    PROC LoadSlot_P06(num slot, VAR bool used, VAR num subType, VAR num toolSel, VAR num lenMM,
                       VAR robtarget arcStart, VAR robtarget arcEnd, VAR robtarget approach, VAR robtarget retract, VAR robtarget trans)
        IF slot = 1 THEN
            used := P06W01_Used;
            subType := P06W01_SubType;
            toolSel := P06W01_ToolSel;
            lenMM := P06W01_LenMM;
            arcStart := P06W01_ArcStart;
            arcEnd := P06W01_ArcEnd;
            approach := P06W01_Approach;
            retract := P06W01_Retract;
            trans := P06W01_Trans;
        ELSEIF slot = 2 THEN
            used := P06W02_Used;
            subType := P06W02_SubType;
            toolSel := P06W02_ToolSel;
            lenMM := P06W02_LenMM;
            arcStart := P06W02_ArcStart;
            arcEnd := P06W02_ArcEnd;
            approach := P06W02_Approach;
            retract := P06W02_Retract;
            trans := P06W02_Trans;
        ELSEIF slot = 3 THEN
            used := P06W03_Used;
            subType := P06W03_SubType;
            toolSel := P06W03_ToolSel;
            lenMM := P06W03_LenMM;
            arcStart := P06W03_ArcStart;
            arcEnd := P06W03_ArcEnd;
            approach := P06W03_Approach;
            retract := P06W03_Retract;
            trans := P06W03_Trans;
        ELSEIF slot = 4 THEN
            used := P06W04_Used;
            subType := P06W04_SubType;
            toolSel := P06W04_ToolSel;
            lenMM := P06W04_LenMM;
            arcStart := P06W04_ArcStart;
            arcEnd := P06W04_ArcEnd;
            approach := P06W04_Approach;
            retract := P06W04_Retract;
            trans := P06W04_Trans;
        ELSEIF slot = 5 THEN
            used := P06W05_Used;
            subType := P06W05_SubType;
            toolSel := P06W05_ToolSel;
            lenMM := P06W05_LenMM;
            arcStart := P06W05_ArcStart;
            arcEnd := P06W05_ArcEnd;
            approach := P06W05_Approach;
            retract := P06W05_Retract;
            trans := P06W05_Trans;
        ELSEIF slot = 6 THEN
            used := P06W06_Used;
            subType := P06W06_SubType;
            toolSel := P06W06_ToolSel;
            lenMM := P06W06_LenMM;
            arcStart := P06W06_ArcStart;
            arcEnd := P06W06_ArcEnd;
            approach := P06W06_Approach;
            retract := P06W06_Retract;
            trans := P06W06_Trans;
        ELSEIF slot = 7 THEN
            used := P06W07_Used;
            subType := P06W07_SubType;
            toolSel := P06W07_ToolSel;
            lenMM := P06W07_LenMM;
            arcStart := P06W07_ArcStart;
            arcEnd := P06W07_ArcEnd;
            approach := P06W07_Approach;
            retract := P06W07_Retract;
            trans := P06W07_Trans;
        ELSEIF slot = 8 THEN
            used := P06W08_Used;
            subType := P06W08_SubType;
            toolSel := P06W08_ToolSel;
            lenMM := P06W08_LenMM;
            arcStart := P06W08_ArcStart;
            arcEnd := P06W08_ArcEnd;
            approach := P06W08_Approach;
            retract := P06W08_Retract;
            trans := P06W08_Trans;
        ELSEIF slot = 9 THEN
            used := P06W09_Used;
            subType := P06W09_SubType;
            toolSel := P06W09_ToolSel;
            lenMM := P06W09_LenMM;
            arcStart := P06W09_ArcStart;
            arcEnd := P06W09_ArcEnd;
            approach := P06W09_Approach;
            retract := P06W09_Retract;
            trans := P06W09_Trans;
        ELSEIF slot = 10 THEN
            used := P06W10_Used;
            subType := P06W10_SubType;
            toolSel := P06W10_ToolSel;
            lenMM := P06W10_LenMM;
            arcStart := P06W10_ArcStart;
            arcEnd := P06W10_ArcEnd;
            approach := P06W10_Approach;
            retract := P06W10_Retract;
            trans := P06W10_Trans;
        ELSEIF slot = 11 THEN
            used := P06W11_Used;
            subType := P06W11_SubType;
            toolSel := P06W11_ToolSel;
            lenMM := P06W11_LenMM;
            arcStart := P06W11_ArcStart;
            arcEnd := P06W11_ArcEnd;
            approach := P06W11_Approach;
            retract := P06W11_Retract;
            trans := P06W11_Trans;
        ELSEIF slot = 12 THEN
            used := P06W12_Used;
            subType := P06W12_SubType;
            toolSel := P06W12_ToolSel;
            lenMM := P06W12_LenMM;
            arcStart := P06W12_ArcStart;
            arcEnd := P06W12_ArcEnd;
            approach := P06W12_Approach;
            retract := P06W12_Retract;
            trans := P06W12_Trans;
        ELSEIF slot = 13 THEN
            used := P06W13_Used;
            subType := P06W13_SubType;
            toolSel := P06W13_ToolSel;
            lenMM := P06W13_LenMM;
            arcStart := P06W13_ArcStart;
            arcEnd := P06W13_ArcEnd;
            approach := P06W13_Approach;
            retract := P06W13_Retract;
            trans := P06W13_Trans;
        ELSEIF slot = 14 THEN
            used := P06W14_Used;
            subType := P06W14_SubType;
            toolSel := P06W14_ToolSel;
            lenMM := P06W14_LenMM;
            arcStart := P06W14_ArcStart;
            arcEnd := P06W14_ArcEnd;
            approach := P06W14_Approach;
            retract := P06W14_Retract;
            trans := P06W14_Trans;
        ELSEIF slot = 15 THEN
            used := P06W15_Used;
            subType := P06W15_SubType;
            toolSel := P06W15_ToolSel;
            lenMM := P06W15_LenMM;
            arcStart := P06W15_ArcStart;
            arcEnd := P06W15_ArcEnd;
            approach := P06W15_Approach;
            retract := P06W15_Retract;
            trans := P06W15_Trans;
        ELSEIF slot = 16 THEN
            used := P06W16_Used;
            subType := P06W16_SubType;
            toolSel := P06W16_ToolSel;
            lenMM := P06W16_LenMM;
            arcStart := P06W16_ArcStart;
            arcEnd := P06W16_ArcEnd;
            approach := P06W16_Approach;
            retract := P06W16_Retract;
            trans := P06W16_Trans;
        ELSEIF slot = 17 THEN
            used := P06W17_Used;
            subType := P06W17_SubType;
            toolSel := P06W17_ToolSel;
            lenMM := P06W17_LenMM;
            arcStart := P06W17_ArcStart;
            arcEnd := P06W17_ArcEnd;
            approach := P06W17_Approach;
            retract := P06W17_Retract;
            trans := P06W17_Trans;
        ELSEIF slot = 18 THEN
            used := P06W18_Used;
            subType := P06W18_SubType;
            toolSel := P06W18_ToolSel;
            lenMM := P06W18_LenMM;
            arcStart := P06W18_ArcStart;
            arcEnd := P06W18_ArcEnd;
            approach := P06W18_Approach;
            retract := P06W18_Retract;
            trans := P06W18_Trans;
        ELSEIF slot = 19 THEN
            used := P06W19_Used;
            subType := P06W19_SubType;
            toolSel := P06W19_ToolSel;
            lenMM := P06W19_LenMM;
            arcStart := P06W19_ArcStart;
            arcEnd := P06W19_ArcEnd;
            approach := P06W19_Approach;
            retract := P06W19_Retract;
            trans := P06W19_Trans;
        ELSEIF slot = 20 THEN
            used := P06W20_Used;
            subType := P06W20_SubType;
            toolSel := P06W20_ToolSel;
            lenMM := P06W20_LenMM;
            arcStart := P06W20_ArcStart;
            arcEnd := P06W20_ArcEnd;
            approach := P06W20_Approach;
            retract := P06W20_Retract;
            trans := P06W20_Trans;
        ELSEIF slot = 21 THEN
            used := P06W21_Used;
            subType := P06W21_SubType;
            toolSel := P06W21_ToolSel;
            lenMM := P06W21_LenMM;
            arcStart := P06W21_ArcStart;
            arcEnd := P06W21_ArcEnd;
            approach := P06W21_Approach;
            retract := P06W21_Retract;
            trans := P06W21_Trans;
        ELSEIF slot = 22 THEN
            used := P06W22_Used;
            subType := P06W22_SubType;
            toolSel := P06W22_ToolSel;
            lenMM := P06W22_LenMM;
            arcStart := P06W22_ArcStart;
            arcEnd := P06W22_ArcEnd;
            approach := P06W22_Approach;
            retract := P06W22_Retract;
            trans := P06W22_Trans;
        ELSEIF slot = 23 THEN
            used := P06W23_Used;
            subType := P06W23_SubType;
            toolSel := P06W23_ToolSel;
            lenMM := P06W23_LenMM;
            arcStart := P06W23_ArcStart;
            arcEnd := P06W23_ArcEnd;
            approach := P06W23_Approach;
            retract := P06W23_Retract;
            trans := P06W23_Trans;
        ELSEIF slot = 24 THEN
            used := P06W24_Used;
            subType := P06W24_SubType;
            toolSel := P06W24_ToolSel;
            lenMM := P06W24_LenMM;
            arcStart := P06W24_ArcStart;
            arcEnd := P06W24_ArcEnd;
            approach := P06W24_Approach;
            retract := P06W24_Retract;
            trans := P06W24_Trans;
        ELSEIF slot = 25 THEN
            used := P06W25_Used;
            subType := P06W25_SubType;
            toolSel := P06W25_ToolSel;
            lenMM := P06W25_LenMM;
            arcStart := P06W25_ArcStart;
            arcEnd := P06W25_ArcEnd;
            approach := P06W25_Approach;
            retract := P06W25_Retract;
            trans := P06W25_Trans;
        ELSEIF slot = 26 THEN
            used := P06W26_Used;
            subType := P06W26_SubType;
            toolSel := P06W26_ToolSel;
            lenMM := P06W26_LenMM;
            arcStart := P06W26_ArcStart;
            arcEnd := P06W26_ArcEnd;
            approach := P06W26_Approach;
            retract := P06W26_Retract;
            trans := P06W26_Trans;
        ELSEIF slot = 27 THEN
            used := P06W27_Used;
            subType := P06W27_SubType;
            toolSel := P06W27_ToolSel;
            lenMM := P06W27_LenMM;
            arcStart := P06W27_ArcStart;
            arcEnd := P06W27_ArcEnd;
            approach := P06W27_Approach;
            retract := P06W27_Retract;
            trans := P06W27_Trans;
        ELSEIF slot = 28 THEN
            used := P06W28_Used;
            subType := P06W28_SubType;
            toolSel := P06W28_ToolSel;
            lenMM := P06W28_LenMM;
            arcStart := P06W28_ArcStart;
            arcEnd := P06W28_ArcEnd;
            approach := P06W28_Approach;
            retract := P06W28_Retract;
            trans := P06W28_Trans;
        ELSEIF slot = 29 THEN
            used := P06W29_Used;
            subType := P06W29_SubType;
            toolSel := P06W29_ToolSel;
            lenMM := P06W29_LenMM;
            arcStart := P06W29_ArcStart;
            arcEnd := P06W29_ArcEnd;
            approach := P06W29_Approach;
            retract := P06W29_Retract;
            trans := P06W29_Trans;
        ELSEIF slot = 30 THEN
            used := P06W30_Used;
            subType := P06W30_SubType;
            toolSel := P06W30_ToolSel;
            lenMM := P06W30_LenMM;
            arcStart := P06W30_ArcStart;
            arcEnd := P06W30_ArcEnd;
            approach := P06W30_Approach;
            retract := P06W30_Retract;
            trans := P06W30_Trans;
        ELSE
            used := FALSE;
        ENDIF
    ENDPROC

    PROC ClearSlot_P06(num slot)
        IF slot = 1 THEN
            P06W01_Used := FALSE;
            P06W01_SubType := 0;
            P06W01_ToolSel := 0;
            P06W01_LenMM := 0;
            P06W01_ArcStart := [[0,0,0],[1,0,0,0],[0,0,0,0],[9E9,9E9,9E9,9E9,9E9,9E9]];
            P06W01_ArcEnd := [[0,0,0],[1,0,0,0],[0,0,0,0],[9E9,9E9,9E9,9E9,9E9,9E9]];
            P06W01_Approach := [[0,0,0],[1,0,0,0],[0,0,0,0],[9E9,9E9,9E9,9E9,9E9,9E9]];
            P06W01_Retract := [[0,0,0],[1,0,0,0],[0,0,0,0],[9E9,9E9,9E9,9E9,9E9,9E9]];
            P06W01_Trans := [[0,0,0],[1,0,0,0],[0,0,0,0],[9E9,9E9,9E9,9E9,9E9,9E9]];
        ELSEIF slot = 2 THEN
            P06W02_Used := FALSE;
            P06W02_SubType := 0;
            P06W02_ToolSel := 0;
            P06W02_LenMM := 0;
            P06W02_ArcStart := [[0,0,0],[1,0,0,0],[0,0,0,0],[9E9,9E9,9E9,9E9,9E9,9E9]];
            P06W02_ArcEnd := [[0,0,0],[1,0,0,0],[0,0,0,0],[9E9,9E9,9E9,9E9,9E9,9E9]];
            P06W02_Approach := [[0,0,0],[1,0,0,0],[0,0,0,0],[9E9,9E9,9E9,9E9,9E9,9E9]];
            P06W02_Retract := [[0,0,0],[1,0,0,0],[0,0,0,0],[9E9,9E9,9E9,9E9,9E9,9E9]];
            P06W02_Trans := [[0,0,0],[1,0,0,0],[0,0,0,0],[9E9,9E9,9E9,9E9,9E9,9E9]];
        ELSEIF slot = 3 THEN
            P06W03_Used := FALSE;
            P06W03_SubType := 0;
            P06W03_ToolSel := 0;
            P06W03_LenMM := 0;
            P06W03_ArcStart := [[0,0,0],[1,0,0,0],[0,0,0,0],[9E9,9E9,9E9,9E9,9E9,9E9]];
            P06W03_ArcEnd := [[0,0,0],[1,0,0,0],[0,0,0,0],[9E9,9E9,9E9,9E9,9E9,9E9]];
            P06W03_Approach := [[0,0,0],[1,0,0,0],[0,0,0,0],[9E9,9E9,9E9,9E9,9E9,9E9]];
            P06W03_Retract := [[0,0,0],[1,0,0,0],[0,0,0,0],[9E9,9E9,9E9,9E9,9E9,9E9]];
            P06W03_Trans := [[0,0,0],[1,0,0,0],[0,0,0,0],[9E9,9E9,9E9,9E9,9E9,9E9]];
        ELSEIF slot = 4 THEN
            P06W04_Used := FALSE;
            P06W04_SubType := 0;
            P06W04_ToolSel := 0;
            P06W04_LenMM := 0;
            P06W04_ArcStart := [[0,0,0],[1,0,0,0],[0,0,0,0],[9E9,9E9,9E9,9E9,9E9,9E9]];
            P06W04_ArcEnd := [[0,0,0],[1,0,0,0],[0,0,0,0],[9E9,9E9,9E9,9E9,9E9,9E9]];
            P06W04_Approach := [[0,0,0],[1,0,0,0],[0,0,0,0],[9E9,9E9,9E9,9E9,9E9,9E9]];
            P06W04_Retract := [[0,0,0],[1,0,0,0],[0,0,0,0],[9E9,9E9,9E9,9E9,9E9,9E9]];
            P06W04_Trans := [[0,0,0],[1,0,0,0],[0,0,0,0],[9E9,9E9,9E9,9E9,9E9,9E9]];
        ELSEIF slot = 5 THEN
            P06W05_Used := FALSE;
            P06W05_SubType := 0;
            P06W05_ToolSel := 0;
            P06W05_LenMM := 0;
            P06W05_ArcStart := [[0,0,0],[1,0,0,0],[0,0,0,0],[9E9,9E9,9E9,9E9,9E9,9E9]];
            P06W05_ArcEnd := [[0,0,0],[1,0,0,0],[0,0,0,0],[9E9,9E9,9E9,9E9,9E9,9E9]];
            P06W05_Approach := [[0,0,0],[1,0,0,0],[0,0,0,0],[9E9,9E9,9E9,9E9,9E9,9E9]];
            P06W05_Retract := [[0,0,0],[1,0,0,0],[0,0,0,0],[9E9,9E9,9E9,9E9,9E9,9E9]];
            P06W05_Trans := [[0,0,0],[1,0,0,0],[0,0,0,0],[9E9,9E9,9E9,9E9,9E9,9E9]];
        ELSEIF slot = 6 THEN
            P06W06_Used := FALSE;
            P06W06_SubType := 0;
            P06W06_ToolSel := 0;
            P06W06_LenMM := 0;
            P06W06_ArcStart := [[0,0,0],[1,0,0,0],[0,0,0,0],[9E9,9E9,9E9,9E9,9E9,9E9]];
            P06W06_ArcEnd := [[0,0,0],[1,0,0,0],[0,0,0,0],[9E9,9E9,9E9,9E9,9E9,9E9]];
            P06W06_Approach := [[0,0,0],[1,0,0,0],[0,0,0,0],[9E9,9E9,9E9,9E9,9E9,9E9]];
            P06W06_Retract := [[0,0,0],[1,0,0,0],[0,0,0,0],[9E9,9E9,9E9,9E9,9E9,9E9]];
            P06W06_Trans := [[0,0,0],[1,0,0,0],[0,0,0,0],[9E9,9E9,9E9,9E9,9E9,9E9]];
        ELSEIF slot = 7 THEN
            P06W07_Used := FALSE;
            P06W07_SubType := 0;
            P06W07_ToolSel := 0;
            P06W07_LenMM := 0;
            P06W07_ArcStart := [[0,0,0],[1,0,0,0],[0,0,0,0],[9E9,9E9,9E9,9E9,9E9,9E9]];
            P06W07_ArcEnd := [[0,0,0],[1,0,0,0],[0,0,0,0],[9E9,9E9,9E9,9E9,9E9,9E9]];
            P06W07_Approach := [[0,0,0],[1,0,0,0],[0,0,0,0],[9E9,9E9,9E9,9E9,9E9,9E9]];
            P06W07_Retract := [[0,0,0],[1,0,0,0],[0,0,0,0],[9E9,9E9,9E9,9E9,9E9,9E9]];
            P06W07_Trans := [[0,0,0],[1,0,0,0],[0,0,0,0],[9E9,9E9,9E9,9E9,9E9,9E9]];
        ELSEIF slot = 8 THEN
            P06W08_Used := FALSE;
            P06W08_SubType := 0;
            P06W08_ToolSel := 0;
            P06W08_LenMM := 0;
            P06W08_ArcStart := [[0,0,0],[1,0,0,0],[0,0,0,0],[9E9,9E9,9E9,9E9,9E9,9E9]];
            P06W08_ArcEnd := [[0,0,0],[1,0,0,0],[0,0,0,0],[9E9,9E9,9E9,9E9,9E9,9E9]];
            P06W08_Approach := [[0,0,0],[1,0,0,0],[0,0,0,0],[9E9,9E9,9E9,9E9,9E9,9E9]];
            P06W08_Retract := [[0,0,0],[1,0,0,0],[0,0,0,0],[9E9,9E9,9E9,9E9,9E9,9E9]];
            P06W08_Trans := [[0,0,0],[1,0,0,0],[0,0,0,0],[9E9,9E9,9E9,9E9,9E9,9E9]];
        ELSEIF slot = 9 THEN
            P06W09_Used := FALSE;
            P06W09_SubType := 0;
            P06W09_ToolSel := 0;
            P06W09_LenMM := 0;
            P06W09_ArcStart := [[0,0,0],[1,0,0,0],[0,0,0,0],[9E9,9E9,9E9,9E9,9E9,9E9]];
            P06W09_ArcEnd := [[0,0,0],[1,0,0,0],[0,0,0,0],[9E9,9E9,9E9,9E9,9E9,9E9]];
            P06W09_Approach := [[0,0,0],[1,0,0,0],[0,0,0,0],[9E9,9E9,9E9,9E9,9E9,9E9]];
            P06W09_Retract := [[0,0,0],[1,0,0,0],[0,0,0,0],[9E9,9E9,9E9,9E9,9E9,9E9]];
            P06W09_Trans := [[0,0,0],[1,0,0,0],[0,0,0,0],[9E9,9E9,9E9,9E9,9E9,9E9]];
        ELSEIF slot = 10 THEN
            P06W10_Used := FALSE;
            P06W10_SubType := 0;
            P06W10_ToolSel := 0;
            P06W10_LenMM := 0;
            P06W10_ArcStart := [[0,0,0],[1,0,0,0],[0,0,0,0],[9E9,9E9,9E9,9E9,9E9,9E9]];
            P06W10_ArcEnd := [[0,0,0],[1,0,0,0],[0,0,0,0],[9E9,9E9,9E9,9E9,9E9,9E9]];
            P06W10_Approach := [[0,0,0],[1,0,0,0],[0,0,0,0],[9E9,9E9,9E9,9E9,9E9,9E9]];
            P06W10_Retract := [[0,0,0],[1,0,0,0],[0,0,0,0],[9E9,9E9,9E9,9E9,9E9,9E9]];
            P06W10_Trans := [[0,0,0],[1,0,0,0],[0,0,0,0],[9E9,9E9,9E9,9E9,9E9,9E9]];
        ELSEIF slot = 11 THEN
            P06W11_Used := FALSE;
            P06W11_SubType := 0;
            P06W11_ToolSel := 0;
            P06W11_LenMM := 0;
            P06W11_ArcStart := [[0,0,0],[1,0,0,0],[0,0,0,0],[9E9,9E9,9E9,9E9,9E9,9E9]];
            P06W11_ArcEnd := [[0,0,0],[1,0,0,0],[0,0,0,0],[9E9,9E9,9E9,9E9,9E9,9E9]];
            P06W11_Approach := [[0,0,0],[1,0,0,0],[0,0,0,0],[9E9,9E9,9E9,9E9,9E9,9E9]];
            P06W11_Retract := [[0,0,0],[1,0,0,0],[0,0,0,0],[9E9,9E9,9E9,9E9,9E9,9E9]];
            P06W11_Trans := [[0,0,0],[1,0,0,0],[0,0,0,0],[9E9,9E9,9E9,9E9,9E9,9E9]];
        ELSEIF slot = 12 THEN
            P06W12_Used := FALSE;
            P06W12_SubType := 0;
            P06W12_ToolSel := 0;
            P06W12_LenMM := 0;
            P06W12_ArcStart := [[0,0,0],[1,0,0,0],[0,0,0,0],[9E9,9E9,9E9,9E9,9E9,9E9]];
            P06W12_ArcEnd := [[0,0,0],[1,0,0,0],[0,0,0,0],[9E9,9E9,9E9,9E9,9E9,9E9]];
            P06W12_Approach := [[0,0,0],[1,0,0,0],[0,0,0,0],[9E9,9E9,9E9,9E9,9E9,9E9]];
            P06W12_Retract := [[0,0,0],[1,0,0,0],[0,0,0,0],[9E9,9E9,9E9,9E9,9E9,9E9]];
            P06W12_Trans := [[0,0,0],[1,0,0,0],[0,0,0,0],[9E9,9E9,9E9,9E9,9E9,9E9]];
        ELSEIF slot = 13 THEN
            P06W13_Used := FALSE;
            P06W13_SubType := 0;
            P06W13_ToolSel := 0;
            P06W13_LenMM := 0;
            P06W13_ArcStart := [[0,0,0],[1,0,0,0],[0,0,0,0],[9E9,9E9,9E9,9E9,9E9,9E9]];
            P06W13_ArcEnd := [[0,0,0],[1,0,0,0],[0,0,0,0],[9E9,9E9,9E9,9E9,9E9,9E9]];
            P06W13_Approach := [[0,0,0],[1,0,0,0],[0,0,0,0],[9E9,9E9,9E9,9E9,9E9,9E9]];
            P06W13_Retract := [[0,0,0],[1,0,0,0],[0,0,0,0],[9E9,9E9,9E9,9E9,9E9,9E9]];
            P06W13_Trans := [[0,0,0],[1,0,0,0],[0,0,0,0],[9E9,9E9,9E9,9E9,9E9,9E9]];
        ELSEIF slot = 14 THEN
            P06W14_Used := FALSE;
            P06W14_SubType := 0;
            P06W14_ToolSel := 0;
            P06W14_LenMM := 0;
            P06W14_ArcStart := [[0,0,0],[1,0,0,0],[0,0,0,0],[9E9,9E9,9E9,9E9,9E9,9E9]];
            P06W14_ArcEnd := [[0,0,0],[1,0,0,0],[0,0,0,0],[9E9,9E9,9E9,9E9,9E9,9E9]];
            P06W14_Approach := [[0,0,0],[1,0,0,0],[0,0,0,0],[9E9,9E9,9E9,9E9,9E9,9E9]];
            P06W14_Retract := [[0,0,0],[1,0,0,0],[0,0,0,0],[9E9,9E9,9E9,9E9,9E9,9E9]];
            P06W14_Trans := [[0,0,0],[1,0,0,0],[0,0,0,0],[9E9,9E9,9E9,9E9,9E9,9E9]];
        ELSEIF slot = 15 THEN
            P06W15_Used := FALSE;
            P06W15_SubType := 0;
            P06W15_ToolSel := 0;
            P06W15_LenMM := 0;
            P06W15_ArcStart := [[0,0,0],[1,0,0,0],[0,0,0,0],[9E9,9E9,9E9,9E9,9E9,9E9]];
            P06W15_ArcEnd := [[0,0,0],[1,0,0,0],[0,0,0,0],[9E9,9E9,9E9,9E9,9E9,9E9]];
            P06W15_Approach := [[0,0,0],[1,0,0,0],[0,0,0,0],[9E9,9E9,9E9,9E9,9E9,9E9]];
            P06W15_Retract := [[0,0,0],[1,0,0,0],[0,0,0,0],[9E9,9E9,9E9,9E9,9E9,9E9]];
            P06W15_Trans := [[0,0,0],[1,0,0,0],[0,0,0,0],[9E9,9E9,9E9,9E9,9E9,9E9]];
        ELSEIF slot = 16 THEN
            P06W16_Used := FALSE;
            P06W16_SubType := 0;
            P06W16_ToolSel := 0;
            P06W16_LenMM := 0;
            P06W16_ArcStart := [[0,0,0],[1,0,0,0],[0,0,0,0],[9E9,9E9,9E9,9E9,9E9,9E9]];
            P06W16_ArcEnd := [[0,0,0],[1,0,0,0],[0,0,0,0],[9E9,9E9,9E9,9E9,9E9,9E9]];
            P06W16_Approach := [[0,0,0],[1,0,0,0],[0,0,0,0],[9E9,9E9,9E9,9E9,9E9,9E9]];
            P06W16_Retract := [[0,0,0],[1,0,0,0],[0,0,0,0],[9E9,9E9,9E9,9E9,9E9,9E9]];
            P06W16_Trans := [[0,0,0],[1,0,0,0],[0,0,0,0],[9E9,9E9,9E9,9E9,9E9,9E9]];
        ELSEIF slot = 17 THEN
            P06W17_Used := FALSE;
            P06W17_SubType := 0;
            P06W17_ToolSel := 0;
            P06W17_LenMM := 0;
            P06W17_ArcStart := [[0,0,0],[1,0,0,0],[0,0,0,0],[9E9,9E9,9E9,9E9,9E9,9E9]];
            P06W17_ArcEnd := [[0,0,0],[1,0,0,0],[0,0,0,0],[9E9,9E9,9E9,9E9,9E9,9E9]];
            P06W17_Approach := [[0,0,0],[1,0,0,0],[0,0,0,0],[9E9,9E9,9E9,9E9,9E9,9E9]];
            P06W17_Retract := [[0,0,0],[1,0,0,0],[0,0,0,0],[9E9,9E9,9E9,9E9,9E9,9E9]];
            P06W17_Trans := [[0,0,0],[1,0,0,0],[0,0,0,0],[9E9,9E9,9E9,9E9,9E9,9E9]];
        ELSEIF slot = 18 THEN
            P06W18_Used := FALSE;
            P06W18_SubType := 0;
            P06W18_ToolSel := 0;
            P06W18_LenMM := 0;
            P06W18_ArcStart := [[0,0,0],[1,0,0,0],[0,0,0,0],[9E9,9E9,9E9,9E9,9E9,9E9]];
            P06W18_ArcEnd := [[0,0,0],[1,0,0,0],[0,0,0,0],[9E9,9E9,9E9,9E9,9E9,9E9]];
            P06W18_Approach := [[0,0,0],[1,0,0,0],[0,0,0,0],[9E9,9E9,9E9,9E9,9E9,9E9]];
            P06W18_Retract := [[0,0,0],[1,0,0,0],[0,0,0,0],[9E9,9E9,9E9,9E9,9E9,9E9]];
            P06W18_Trans := [[0,0,0],[1,0,0,0],[0,0,0,0],[9E9,9E9,9E9,9E9,9E9,9E9]];
        ELSEIF slot = 19 THEN
            P06W19_Used := FALSE;
            P06W19_SubType := 0;
            P06W19_ToolSel := 0;
            P06W19_LenMM := 0;
            P06W19_ArcStart := [[0,0,0],[1,0,0,0],[0,0,0,0],[9E9,9E9,9E9,9E9,9E9,9E9]];
            P06W19_ArcEnd := [[0,0,0],[1,0,0,0],[0,0,0,0],[9E9,9E9,9E9,9E9,9E9,9E9]];
            P06W19_Approach := [[0,0,0],[1,0,0,0],[0,0,0,0],[9E9,9E9,9E9,9E9,9E9,9E9]];
            P06W19_Retract := [[0,0,0],[1,0,0,0],[0,0,0,0],[9E9,9E9,9E9,9E9,9E9,9E9]];
            P06W19_Trans := [[0,0,0],[1,0,0,0],[0,0,0,0],[9E9,9E9,9E9,9E9,9E9,9E9]];
        ELSEIF slot = 20 THEN
            P06W20_Used := FALSE;
            P06W20_SubType := 0;
            P06W20_ToolSel := 0;
            P06W20_LenMM := 0;
            P06W20_ArcStart := [[0,0,0],[1,0,0,0],[0,0,0,0],[9E9,9E9,9E9,9E9,9E9,9E9]];
            P06W20_ArcEnd := [[0,0,0],[1,0,0,0],[0,0,0,0],[9E9,9E9,9E9,9E9,9E9,9E9]];
            P06W20_Approach := [[0,0,0],[1,0,0,0],[0,0,0,0],[9E9,9E9,9E9,9E9,9E9,9E9]];
            P06W20_Retract := [[0,0,0],[1,0,0,0],[0,0,0,0],[9E9,9E9,9E9,9E9,9E9,9E9]];
            P06W20_Trans := [[0,0,0],[1,0,0,0],[0,0,0,0],[9E9,9E9,9E9,9E9,9E9,9E9]];
        ELSEIF slot = 21 THEN
            P06W21_Used := FALSE;
            P06W21_SubType := 0;
            P06W21_ToolSel := 0;
            P06W21_LenMM := 0;
            P06W21_ArcStart := [[0,0,0],[1,0,0,0],[0,0,0,0],[9E9,9E9,9E9,9E9,9E9,9E9]];
            P06W21_ArcEnd := [[0,0,0],[1,0,0,0],[0,0,0,0],[9E9,9E9,9E9,9E9,9E9,9E9]];
            P06W21_Approach := [[0,0,0],[1,0,0,0],[0,0,0,0],[9E9,9E9,9E9,9E9,9E9,9E9]];
            P06W21_Retract := [[0,0,0],[1,0,0,0],[0,0,0,0],[9E9,9E9,9E9,9E9,9E9,9E9]];
            P06W21_Trans := [[0,0,0],[1,0,0,0],[0,0,0,0],[9E9,9E9,9E9,9E9,9E9,9E9]];
        ELSEIF slot = 22 THEN
            P06W22_Used := FALSE;
            P06W22_SubType := 0;
            P06W22_ToolSel := 0;
            P06W22_LenMM := 0;
            P06W22_ArcStart := [[0,0,0],[1,0,0,0],[0,0,0,0],[9E9,9E9,9E9,9E9,9E9,9E9]];
            P06W22_ArcEnd := [[0,0,0],[1,0,0,0],[0,0,0,0],[9E9,9E9,9E9,9E9,9E9,9E9]];
            P06W22_Approach := [[0,0,0],[1,0,0,0],[0,0,0,0],[9E9,9E9,9E9,9E9,9E9,9E9]];
            P06W22_Retract := [[0,0,0],[1,0,0,0],[0,0,0,0],[9E9,9E9,9E9,9E9,9E9,9E9]];
            P06W22_Trans := [[0,0,0],[1,0,0,0],[0,0,0,0],[9E9,9E9,9E9,9E9,9E9,9E9]];
        ELSEIF slot = 23 THEN
            P06W23_Used := FALSE;
            P06W23_SubType := 0;
            P06W23_ToolSel := 0;
            P06W23_LenMM := 0;
            P06W23_ArcStart := [[0,0,0],[1,0,0,0],[0,0,0,0],[9E9,9E9,9E9,9E9,9E9,9E9]];
            P06W23_ArcEnd := [[0,0,0],[1,0,0,0],[0,0,0,0],[9E9,9E9,9E9,9E9,9E9,9E9]];
            P06W23_Approach := [[0,0,0],[1,0,0,0],[0,0,0,0],[9E9,9E9,9E9,9E9,9E9,9E9]];
            P06W23_Retract := [[0,0,0],[1,0,0,0],[0,0,0,0],[9E9,9E9,9E9,9E9,9E9,9E9]];
            P06W23_Trans := [[0,0,0],[1,0,0,0],[0,0,0,0],[9E9,9E9,9E9,9E9,9E9,9E9]];
        ELSEIF slot = 24 THEN
            P06W24_Used := FALSE;
            P06W24_SubType := 0;
            P06W24_ToolSel := 0;
            P06W24_LenMM := 0;
            P06W24_ArcStart := [[0,0,0],[1,0,0,0],[0,0,0,0],[9E9,9E9,9E9,9E9,9E9,9E9]];
            P06W24_ArcEnd := [[0,0,0],[1,0,0,0],[0,0,0,0],[9E9,9E9,9E9,9E9,9E9,9E9]];
            P06W24_Approach := [[0,0,0],[1,0,0,0],[0,0,0,0],[9E9,9E9,9E9,9E9,9E9,9E9]];
            P06W24_Retract := [[0,0,0],[1,0,0,0],[0,0,0,0],[9E9,9E9,9E9,9E9,9E9,9E9]];
            P06W24_Trans := [[0,0,0],[1,0,0,0],[0,0,0,0],[9E9,9E9,9E9,9E9,9E9,9E9]];
        ELSEIF slot = 25 THEN
            P06W25_Used := FALSE;
            P06W25_SubType := 0;
            P06W25_ToolSel := 0;
            P06W25_LenMM := 0;
            P06W25_ArcStart := [[0,0,0],[1,0,0,0],[0,0,0,0],[9E9,9E9,9E9,9E9,9E9,9E9]];
            P06W25_ArcEnd := [[0,0,0],[1,0,0,0],[0,0,0,0],[9E9,9E9,9E9,9E9,9E9,9E9]];
            P06W25_Approach := [[0,0,0],[1,0,0,0],[0,0,0,0],[9E9,9E9,9E9,9E9,9E9,9E9]];
            P06W25_Retract := [[0,0,0],[1,0,0,0],[0,0,0,0],[9E9,9E9,9E9,9E9,9E9,9E9]];
            P06W25_Trans := [[0,0,0],[1,0,0,0],[0,0,0,0],[9E9,9E9,9E9,9E9,9E9,9E9]];
        ELSEIF slot = 26 THEN
            P06W26_Used := FALSE;
            P06W26_SubType := 0;
            P06W26_ToolSel := 0;
            P06W26_LenMM := 0;
            P06W26_ArcStart := [[0,0,0],[1,0,0,0],[0,0,0,0],[9E9,9E9,9E9,9E9,9E9,9E9]];
            P06W26_ArcEnd := [[0,0,0],[1,0,0,0],[0,0,0,0],[9E9,9E9,9E9,9E9,9E9,9E9]];
            P06W26_Approach := [[0,0,0],[1,0,0,0],[0,0,0,0],[9E9,9E9,9E9,9E9,9E9,9E9]];
            P06W26_Retract := [[0,0,0],[1,0,0,0],[0,0,0,0],[9E9,9E9,9E9,9E9,9E9,9E9]];
            P06W26_Trans := [[0,0,0],[1,0,0,0],[0,0,0,0],[9E9,9E9,9E9,9E9,9E9,9E9]];
        ELSEIF slot = 27 THEN
            P06W27_Used := FALSE;
            P06W27_SubType := 0;
            P06W27_ToolSel := 0;
            P06W27_LenMM := 0;
            P06W27_ArcStart := [[0,0,0],[1,0,0,0],[0,0,0,0],[9E9,9E9,9E9,9E9,9E9,9E9]];
            P06W27_ArcEnd := [[0,0,0],[1,0,0,0],[0,0,0,0],[9E9,9E9,9E9,9E9,9E9,9E9]];
            P06W27_Approach := [[0,0,0],[1,0,0,0],[0,0,0,0],[9E9,9E9,9E9,9E9,9E9,9E9]];
            P06W27_Retract := [[0,0,0],[1,0,0,0],[0,0,0,0],[9E9,9E9,9E9,9E9,9E9,9E9]];
            P06W27_Trans := [[0,0,0],[1,0,0,0],[0,0,0,0],[9E9,9E9,9E9,9E9,9E9,9E9]];
        ELSEIF slot = 28 THEN
            P06W28_Used := FALSE;
            P06W28_SubType := 0;
            P06W28_ToolSel := 0;
            P06W28_LenMM := 0;
            P06W28_ArcStart := [[0,0,0],[1,0,0,0],[0,0,0,0],[9E9,9E9,9E9,9E9,9E9,9E9]];
            P06W28_ArcEnd := [[0,0,0],[1,0,0,0],[0,0,0,0],[9E9,9E9,9E9,9E9,9E9,9E9]];
            P06W28_Approach := [[0,0,0],[1,0,0,0],[0,0,0,0],[9E9,9E9,9E9,9E9,9E9,9E9]];
            P06W28_Retract := [[0,0,0],[1,0,0,0],[0,0,0,0],[9E9,9E9,9E9,9E9,9E9,9E9]];
            P06W28_Trans := [[0,0,0],[1,0,0,0],[0,0,0,0],[9E9,9E9,9E9,9E9,9E9,9E9]];
        ELSEIF slot = 29 THEN
            P06W29_Used := FALSE;
            P06W29_SubType := 0;
            P06W29_ToolSel := 0;
            P06W29_LenMM := 0;
            P06W29_ArcStart := [[0,0,0],[1,0,0,0],[0,0,0,0],[9E9,9E9,9E9,9E9,9E9,9E9]];
            P06W29_ArcEnd := [[0,0,0],[1,0,0,0],[0,0,0,0],[9E9,9E9,9E9,9E9,9E9,9E9]];
            P06W29_Approach := [[0,0,0],[1,0,0,0],[0,0,0,0],[9E9,9E9,9E9,9E9,9E9,9E9]];
            P06W29_Retract := [[0,0,0],[1,0,0,0],[0,0,0,0],[9E9,9E9,9E9,9E9,9E9,9E9]];
            P06W29_Trans := [[0,0,0],[1,0,0,0],[0,0,0,0],[9E9,9E9,9E9,9E9,9E9,9E9]];
        ELSEIF slot = 30 THEN
            P06W30_Used := FALSE;
            P06W30_SubType := 0;
            P06W30_ToolSel := 0;
            P06W30_LenMM := 0;
            P06W30_ArcStart := [[0,0,0],[1,0,0,0],[0,0,0,0],[9E9,9E9,9E9,9E9,9E9,9E9]];
            P06W30_ArcEnd := [[0,0,0],[1,0,0,0],[0,0,0,0],[9E9,9E9,9E9,9E9,9E9,9E9]];
            P06W30_Approach := [[0,0,0],[1,0,0,0],[0,0,0,0],[9E9,9E9,9E9,9E9,9E9,9E9]];
            P06W30_Retract := [[0,0,0],[1,0,0,0],[0,0,0,0],[9E9,9E9,9E9,9E9,9E9,9E9]];
            P06W30_Trans := [[0,0,0],[1,0,0,0],[0,0,0,0],[9E9,9E9,9E9,9E9,9E9,9E9]];
        ELSE
            TPWrite "Invalid weld slot.";
        ENDIF
    ENDPROC

    PROC StoreNextFree_P06(num subType, num toolSel, num lenMM,
                       robtarget arcStart, robtarget arcEnd, robtarget approach, robtarget retract, robtarget trans)
        IF NOT P06W01_Used THEN
            StoreSlot_P06 1, subType, toolSel, lenMM, arcStart, arcEnd, approach, retract, trans;
            nWeldsP06 := nWeldsP06 + 1;
            RETURN;
        ELSEIF NOT P06W02_Used THEN
            StoreSlot_P06 2, subType, toolSel, lenMM, arcStart, arcEnd, approach, retract, trans;
            nWeldsP06 := nWeldsP06 + 1;
            RETURN;
        ELSEIF NOT P06W03_Used THEN
            StoreSlot_P06 3, subType, toolSel, lenMM, arcStart, arcEnd, approach, retract, trans;
            nWeldsP06 := nWeldsP06 + 1;
            RETURN;
        ELSEIF NOT P06W04_Used THEN
            StoreSlot_P06 4, subType, toolSel, lenMM, arcStart, arcEnd, approach, retract, trans;
            nWeldsP06 := nWeldsP06 + 1;
            RETURN;
        ELSEIF NOT P06W05_Used THEN
            StoreSlot_P06 5, subType, toolSel, lenMM, arcStart, arcEnd, approach, retract, trans;
            nWeldsP06 := nWeldsP06 + 1;
            RETURN;
        ELSEIF NOT P06W06_Used THEN
            StoreSlot_P06 6, subType, toolSel, lenMM, arcStart, arcEnd, approach, retract, trans;
            nWeldsP06 := nWeldsP06 + 1;
            RETURN;
        ELSEIF NOT P06W07_Used THEN
            StoreSlot_P06 7, subType, toolSel, lenMM, arcStart, arcEnd, approach, retract, trans;
            nWeldsP06 := nWeldsP06 + 1;
            RETURN;
        ELSEIF NOT P06W08_Used THEN
            StoreSlot_P06 8, subType, toolSel, lenMM, arcStart, arcEnd, approach, retract, trans;
            nWeldsP06 := nWeldsP06 + 1;
            RETURN;
        ELSEIF NOT P06W09_Used THEN
            StoreSlot_P06 9, subType, toolSel, lenMM, arcStart, arcEnd, approach, retract, trans;
            nWeldsP06 := nWeldsP06 + 1;
            RETURN;
        ELSEIF NOT P06W10_Used THEN
            StoreSlot_P06 10, subType, toolSel, lenMM, arcStart, arcEnd, approach, retract, trans;
            nWeldsP06 := nWeldsP06 + 1;
            RETURN;
        ELSEIF NOT P06W11_Used THEN
            StoreSlot_P06 11, subType, toolSel, lenMM, arcStart, arcEnd, approach, retract, trans;
            nWeldsP06 := nWeldsP06 + 1;
            RETURN;
        ELSEIF NOT P06W12_Used THEN
            StoreSlot_P06 12, subType, toolSel, lenMM, arcStart, arcEnd, approach, retract, trans;
            nWeldsP06 := nWeldsP06 + 1;
            RETURN;
        ELSEIF NOT P06W13_Used THEN
            StoreSlot_P06 13, subType, toolSel, lenMM, arcStart, arcEnd, approach, retract, trans;
            nWeldsP06 := nWeldsP06 + 1;
            RETURN;
        ELSEIF NOT P06W14_Used THEN
            StoreSlot_P06 14, subType, toolSel, lenMM, arcStart, arcEnd, approach, retract, trans;
            nWeldsP06 := nWeldsP06 + 1;
            RETURN;
        ELSEIF NOT P06W15_Used THEN
            StoreSlot_P06 15, subType, toolSel, lenMM, arcStart, arcEnd, approach, retract, trans;
            nWeldsP06 := nWeldsP06 + 1;
            RETURN;
        ELSEIF NOT P06W16_Used THEN
            StoreSlot_P06 16, subType, toolSel, lenMM, arcStart, arcEnd, approach, retract, trans;
            nWeldsP06 := nWeldsP06 + 1;
            RETURN;
        ELSEIF NOT P06W17_Used THEN
            StoreSlot_P06 17, subType, toolSel, lenMM, arcStart, arcEnd, approach, retract, trans;
            nWeldsP06 := nWeldsP06 + 1;
            RETURN;
        ELSEIF NOT P06W18_Used THEN
            StoreSlot_P06 18, subType, toolSel, lenMM, arcStart, arcEnd, approach, retract, trans;
            nWeldsP06 := nWeldsP06 + 1;
            RETURN;
        ELSEIF NOT P06W19_Used THEN
            StoreSlot_P06 19, subType, toolSel, lenMM, arcStart, arcEnd, approach, retract, trans;
            nWeldsP06 := nWeldsP06 + 1;
            RETURN;
        ELSEIF NOT P06W20_Used THEN
            StoreSlot_P06 20, subType, toolSel, lenMM, arcStart, arcEnd, approach, retract, trans;
            nWeldsP06 := nWeldsP06 + 1;
            RETURN;
        ELSEIF NOT P06W21_Used THEN
            StoreSlot_P06 21, subType, toolSel, lenMM, arcStart, arcEnd, approach, retract, trans;
            nWeldsP06 := nWeldsP06 + 1;
            RETURN;
        ELSEIF NOT P06W22_Used THEN
            StoreSlot_P06 22, subType, toolSel, lenMM, arcStart, arcEnd, approach, retract, trans;
            nWeldsP06 := nWeldsP06 + 1;
            RETURN;
        ELSEIF NOT P06W23_Used THEN
            StoreSlot_P06 23, subType, toolSel, lenMM, arcStart, arcEnd, approach, retract, trans;
            nWeldsP06 := nWeldsP06 + 1;
            RETURN;
        ELSEIF NOT P06W24_Used THEN
            StoreSlot_P06 24, subType, toolSel, lenMM, arcStart, arcEnd, approach, retract, trans;
            nWeldsP06 := nWeldsP06 + 1;
            RETURN;
        ELSEIF NOT P06W25_Used THEN
            StoreSlot_P06 25, subType, toolSel, lenMM, arcStart, arcEnd, approach, retract, trans;
            nWeldsP06 := nWeldsP06 + 1;
            RETURN;
        ELSEIF NOT P06W26_Used THEN
            StoreSlot_P06 26, subType, toolSel, lenMM, arcStart, arcEnd, approach, retract, trans;
            nWeldsP06 := nWeldsP06 + 1;
            RETURN;
        ELSEIF NOT P06W27_Used THEN
            StoreSlot_P06 27, subType, toolSel, lenMM, arcStart, arcEnd, approach, retract, trans;
            nWeldsP06 := nWeldsP06 + 1;
            RETURN;
        ELSEIF NOT P06W28_Used THEN
            StoreSlot_P06 28, subType, toolSel, lenMM, arcStart, arcEnd, approach, retract, trans;
            nWeldsP06 := nWeldsP06 + 1;
            RETURN;
        ELSEIF NOT P06W29_Used THEN
            StoreSlot_P06 29, subType, toolSel, lenMM, arcStart, arcEnd, approach, retract, trans;
            nWeldsP06 := nWeldsP06 + 1;
            RETURN;
        ELSEIF NOT P06W30_Used THEN
            StoreSlot_P06 30, subType, toolSel, lenMM, arcStart, arcEnd, approach, retract, trans;
            nWeldsP06 := nWeldsP06 + 1;
            RETURN;
        ELSE
            TPWrite "No free weld slots available.";
        ENDIF
    ENDPROC

    PROC StoreNextFree(num partNum, num subType, num toolSel, num lenMM,
                       robtarget arcStart, robtarget arcEnd, robtarget approach, robtarget retract, robtarget trans)
        IF partNum = 1 THEN
            StoreNextFree_P01 subType, toolSel, lenMM, arcStart, arcEnd, approach, retract, trans;
        ELSEIF partNum = 2 THEN
            StoreNextFree_P02 subType, toolSel, lenMM, arcStart, arcEnd, approach, retract, trans;
        ELSEIF partNum = 3 THEN
            StoreNextFree_P03 subType, toolSel, lenMM, arcStart, arcEnd, approach, retract, trans;
        ELSEIF partNum = 4 THEN
            StoreNextFree_P04 subType, toolSel, lenMM, arcStart, arcEnd, approach, retract, trans;
        ELSEIF partNum = 5 THEN
            StoreNextFree_P05 subType, toolSel, lenMM, arcStart, arcEnd, approach, retract, trans;
        ELSEIF partNum = 6 THEN
            StoreNextFree_P06 subType, toolSel, lenMM, arcStart, arcEnd, approach, retract, trans;
        ELSE
            TPWrite "Invalid part selection.";
        ENDIF
    ENDPROC

    PROC StoreSlot(num partNum, num slot, num subType, num toolSel, num lenMM,
                       robtarget arcStart, robtarget arcEnd, robtarget approach, robtarget retract, robtarget trans)
        IF partNum = 1 THEN
            StoreSlot_P01 slot, subType, toolSel, lenMM, arcStart, arcEnd, approach, retract, trans;
        ELSEIF partNum = 2 THEN
            StoreSlot_P02 slot, subType, toolSel, lenMM, arcStart, arcEnd, approach, retract, trans;
        ELSEIF partNum = 3 THEN
            StoreSlot_P03 slot, subType, toolSel, lenMM, arcStart, arcEnd, approach, retract, trans;
        ELSEIF partNum = 4 THEN
            StoreSlot_P04 slot, subType, toolSel, lenMM, arcStart, arcEnd, approach, retract, trans;
        ELSEIF partNum = 5 THEN
            StoreSlot_P05 slot, subType, toolSel, lenMM, arcStart, arcEnd, approach, retract, trans;
        ELSEIF partNum = 6 THEN
            StoreSlot_P06 slot, subType, toolSel, lenMM, arcStart, arcEnd, approach, retract, trans;
        ELSE
            TPWrite "Invalid part selection.";
        ENDIF
    ENDPROC

    PROC LoadSlot(num partNum, num slot, VAR bool used, VAR num subType, VAR num toolSel, VAR num lenMM,
                       VAR robtarget arcStart, VAR robtarget arcEnd, VAR robtarget approach, VAR robtarget retract, VAR robtarget trans)
        IF partNum = 1 THEN
            LoadSlot_P01 slot, used, subType, toolSel, lenMM, arcStart, arcEnd, approach, retract, trans;
        ELSEIF partNum = 2 THEN
            LoadSlot_P02 slot, used, subType, toolSel, lenMM, arcStart, arcEnd, approach, retract, trans;
        ELSEIF partNum = 3 THEN
            LoadSlot_P03 slot, used, subType, toolSel, lenMM, arcStart, arcEnd, approach, retract, trans;
        ELSEIF partNum = 4 THEN
            LoadSlot_P04 slot, used, subType, toolSel, lenMM, arcStart, arcEnd, approach, retract, trans;
        ELSEIF partNum = 5 THEN
            LoadSlot_P05 slot, used, subType, toolSel, lenMM, arcStart, arcEnd, approach, retract, trans;
        ELSEIF partNum = 6 THEN
            LoadSlot_P06 slot, used, subType, toolSel, lenMM, arcStart, arcEnd, approach, retract, trans;
        ELSE
            used := FALSE;
        ENDIF
    ENDPROC

    PROC ClearSlot(num partNum, num slot)
        IF partNum = 1 THEN
            ClearSlot_P01 slot;
        ELSEIF partNum = 2 THEN
            ClearSlot_P02 slot;
        ELSEIF partNum = 3 THEN
            ClearSlot_P03 slot;
        ELSEIF partNum = 4 THEN
            ClearSlot_P04 slot;
        ELSEIF partNum = 5 THEN
            ClearSlot_P05 slot;
        ELSEIF partNum = 6 THEN
            ClearSlot_P06 slot;
        ELSE
            TPWrite "Invalid part selection.";
        ENDIF
    ENDPROC

    PROC AddWeld(num partNum)
        VAR num major;
        VAR num subType;
        VAR num toolSel;
        VAR num lenIn;
        VAR num lenMM;
        VAR robtarget pStart;
        VAR robtarget pEnd;
        VAR robtarget aS;
        VAR robtarget aE;
        VAR robtarget aA;
        VAR robtarget aR;
        VAR robtarget aT;
        VAR bool repeat;
        VAR num distIn;
        VAR num distMM;
        VAR num cornerType;

        TPWrite "Add Weld - choose type: 1=Vert 2=Horiz 3=Corner 4=Free";
        TPReadNum major, "";

        IF major = WT_VERT THEN
            TPWrite "Vert subtype: 11=YLeft 12=YRight 13=YMid";
            TPReadNum subType, "";
            IF subType = WSV_YLEFT THEN
                toolSel := T_OLEFT;
            ELSEIF subType = WSV_YRIGHT THEN
                toolSel := T_ORIGHT;
            ELSE
                toolSel := T_OYMID;
            ENDIF
        ELSEIF major = WT_HORIZ THEN
            TPWrite "Horiz subtype: 21=XUp 22=XDn 23=XMid";
            TPReadNum subType, "";
            IF subType = WSH_XUP THEN
                toolSel := T_OUP;
            ELSEIF subType = WSH_XDN THEN
                toolSel := T_ODOWN;
            ELSE
                toolSel := T_OXMID;
            ENDIF
        ELSEIF major = WT_FREE THEN
            subType := WSF_FREE;
            TPWrite "Free weld orientation tool: 1=Left 2=Right 3=Up 4=Down 5=YMid 6=XMid";
            TPReadNum toolSel, "";
        ELSE
            TPWrite "Corner subtype: 31=ULC 32=URC 33=DLC 34=DRC";
            TPReadNum subType, "";
            cornerType := subType;
        ENDIF

        IF major = WT_CORNER THEN
            TPWrite "Enter corner length (inches):";
            TPReadNum lenIn, "";
            lenMM := lenIn*INCH;
            TPWrite "Jog to CORNER point (not start). Press Play.";
            Stop;
            pStart := CRobT(\Tool:=tWeldGun);

            ! ---- Y leg ----
            IF cornerType = WSC_ULC OR cornerType = WSC_DLC THEN
                toolSel := T_OLEFT;
                subType := WSV_YLEFT;
            ELSE
                toolSel := T_ORIGHT;
                subType := WSV_YRIGHT;
            ENDIF

            IF cornerType = WSC_DLC OR cornerType = WSC_DRC THEN
                aS := Offs(pStart, 0, +lenMM, 0);
            ELSE
                aS := pStart;
            ENDIF

            BuildWeldFromStart aS, pEnd, subType, toolSel, lenMM, aS, aE, aA, aR, aT;
            StoreNextFree partNum, subType, toolSel, lenMM, aS, aE, aA, aR, aT;
            DryRun aT, aA, aS, aE, aR;

            ! ---- X leg ----
            IF cornerType = WSC_ULC OR cornerType = WSC_URC THEN
                toolSel := T_OUP;
                subType := WSH_XUP;
            ELSE
                toolSel := T_ODOWN;
                subType := WSH_XDN;
            ENDIF

            IF cornerType = WSC_URC OR cornerType = WSC_DRC THEN
                aS := Offs(pStart, -lenMM, 0, 0);
            ELSE
                aS := pStart;
            ENDIF

            BuildWeldFromStart aS, pEnd, subType, toolSel, lenMM, aS, aE, aA, aR, aT;
            StoreNextFree partNum, subType, toolSel, lenMM, aS, aE, aA, aR, aT;
            DryRun aT, aA, aS, aE, aR;
            RETURN;
        ENDIF

        IF major <> WT_FREE THEN
            TPWrite "Enter weld length (inches):";
            TPReadNum lenIn, "";
            lenMM := lenIn*INCH;
        ELSE
            lenMM := 0;
        ENDIF

        IF major = WT_FREE THEN
            TPWrite "Jog to FREE WELD START. Press Play.";
            Stop;
            pStart := CRobT(\Tool:=tWeldGun);
            TPWrite "Jog to FREE WELD END. Press Play.";
            Stop;
            pEnd := CRobT(\Tool:=tWeldGun);
        ELSE
            TPWrite "Jog to START point. Press Play.";
            Stop;
            pStart := CRobT(\Tool:=tWeldGun);
            pEnd := pStart;
        ENDIF

        BuildWeldFromStart pStart, pEnd, subType, toolSel, lenMM, aS, aE, aA, aR, aT;
        StoreNextFree partNum, subType, toolSel, lenMM, aS, aE, aA, aR, aT;
        DryRun aT, aA, aS, aE, aR;

        IF major = WT_VERT OR major = WT_HORIZ THEN
            TPWrite "Repeat? 1=Yes 0=No";
            TPReadNum lenIn, "";
            repeat := (lenIn = 1);
            WHILE repeat DO
                TPWrite "Enter distance to next start (inches, +/-):";
                TPReadNum distIn, "";
                distMM := distIn*INCH;
                IF major = WT_VERT THEN
                    pStart := Offs(pStart, 0, distMM, 0);
                ELSE
                    pStart := Offs(pStart, distMM, 0, 0);
                ENDIF
                BuildWeldFromStart pStart, pEnd, subType, toolSel, lenMM, aS, aE, aA, aR, aT;
                StoreNextFree partNum, subType, toolSel, lenMM, aS, aE, aA, aR, aT;
                DryRun aT, aA, aS, aE, aR;
                TPWrite "Repeat again? 1=Yes 0=No";
                TPReadNum lenIn, "";
                repeat := (lenIn = 1);
            ENDWHILE
        ENDIF
    ENDPROC

    PROC ReviewWeld(num partNum, num slot)
        VAR bool used;
        VAR num subType;
        VAR num toolSel;
        VAR num lenMM;
        VAR robtarget arcStart;
        VAR robtarget arcEnd;
        VAR robtarget approach;
        VAR robtarget retract;
        VAR robtarget trans;
        LoadSlot partNum, slot, used, subType, toolSel, lenMM, arcStart, arcEnd, approach, retract, trans;
        IF used THEN
            DryRun trans, approach, arcStart, arcEnd, retract;
        ELSE
            TPWrite "Slot is empty.";
        ENDIF
    ENDPROC

    PROC EditWeld(num partNum, num slot)
        VAR bool used;
        VAR num subType;
        VAR num toolSel;
        VAR num lenMM;
        VAR num lenIn;
        VAR robtarget arcStart;
        VAR robtarget arcEnd;
        VAR robtarget approach;
        VAR robtarget retract;
        VAR robtarget trans;
        VAR robtarget pStart;
        VAR robtarget pEnd;
        LoadSlot partNum, slot, used, subType, toolSel, lenMM, arcStart, arcEnd, approach, retract, trans;
        IF NOT used THEN
            TPWrite "Slot is empty.";
            RETURN;
        ENDIF
        MoveL approach, v100, z10, tWeldGun;
        TPWrite "Jog to new start point, then press Play.";
        Stop;
        pStart := CRobT(\Tool:=tWeldGun);
        IF subType = WSF_FREE THEN
            TPWrite "Jog to new end point, then press Play.";
            Stop;
            pEnd := CRobT(\Tool:=tWeldGun);
        ELSE
            pEnd := pStart;
        ENDIF
        IF subType <> WSF_FREE THEN
            TPWrite "Enter length (inches) to keep or update:";
            TPReadNum lenIn, "";
            lenMM := lenIn*INCH;
        ENDIF
        BuildWeldFromStart pStart, pEnd, subType, toolSel, lenMM, arcStart, arcEnd, approach, retract, trans;
        StoreSlot partNum, slot, subType, toolSel, lenMM, arcStart, arcEnd, approach, retract, trans;
        TPWrite "Weld updated.";
    ENDPROC

    PROC DeleteWeld(num partNum, num slot)
        VAR num confirm;
        TPWrite "Delete weld slot? 1=Yes 0=No";
        TPReadNum confirm, "";
        IF confirm = 1 THEN
            ClearSlot partNum, slot;
            TPWrite "Weld deleted.";
        ENDIF
    ENDPROC

    PROC mainweld()
        VAR num partNum;
        VAR num choice;
        EnsurePartFrame 1;
        TPWrite "Select Part (1-6):";
        TPReadNum partNum, "";
        TPWrite "1=Teach Ori 2=Setup Part 3=Add Weld 4=Review 5=Edit 6=Delete";
        TPReadNum choice, "";
        IF choice = 1 THEN
            TPWrite "Tool: 1=Left 2=Right 3=Up 4=Down 5=YMid 6=XMid";
            TPReadNum choice, "";
            TeachOrientation choice;
        ELSEIF choice = 2 THEN
            IF partNum = 1 THEN
                SetupP01;
            ELSEIF partNum = 2 THEN
                SetupP02;
            ELSEIF partNum = 3 THEN
                SetupP03;
            ELSEIF partNum = 4 THEN
                SetupP04;
            ELSEIF partNum = 5 THEN
                SetupP05;
            ELSEIF partNum = 6 THEN
                SetupP06;
            ELSE
                TPWrite "Invalid part selection.";
            ENDIF
        ELSEIF choice = 3 THEN
            EnsurePartFrame partNum;
            AddWeld partNum;
        ELSEIF choice = 4 THEN
            EnsurePartFrame partNum;
            TPWrite "Enter weld slot to review (1-30):";
            TPReadNum choice, "";
            ReviewWeld partNum, choice;
        ELSEIF choice = 5 THEN
            EnsurePartFrame partNum;
            TPWrite "Enter weld slot to edit (1-30):";
            TPReadNum choice, "";
            EditWeld partNum, choice;
        ELSEIF choice = 6 THEN
            EnsurePartFrame partNum;
            TPWrite "Enter weld slot to delete (1-30):";
            TPReadNum choice, "";
            DeleteWeld partNum, choice;
        ELSE
            TPWrite "Invalid selection.";
        ENDIF
    ENDPROC

ENDMODULE
